% RSLogix 500 project Batch Part Counter.RSS, saved by version 8.30.00.16 %
PROJECT "UNTITLED"    % processor: Bul.1763 MicroLogix 1100 Series B %

PROGRAM FILES
  LAD 2 "MAIN"  7 rungs
  LAD 3 "IO"  5 rungs

DATA FILES
  O0 OUTPUT  5 elements
  I1 INPUT  7 elements
  S2 STATUS  66 elements
  B3 BINARY  1 elements
  T4 TIMER  1 elements
  C5 COUNTER  1 elements
  R6 CONTROL  1 elements
  N7 INTEGER  1 elements
  F8 FLOAT  1 elements

LADDER 2 "MAIN"
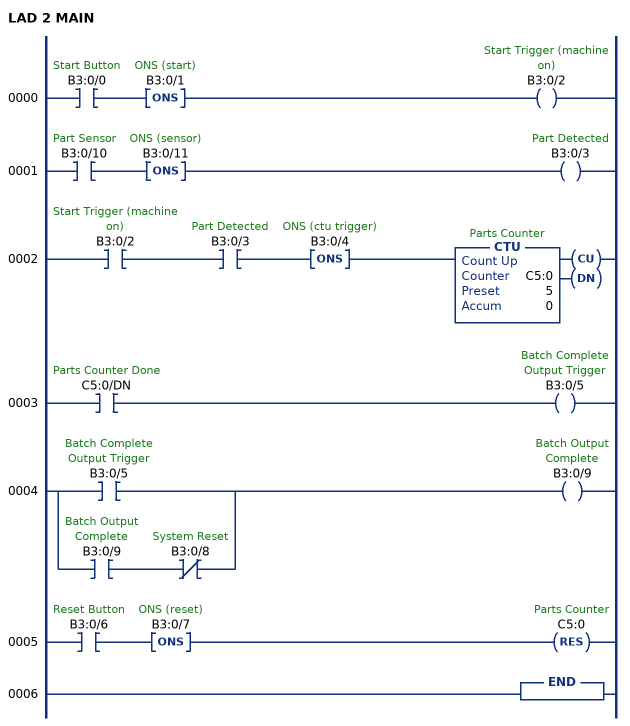
% Rung: 0 %
SOR XIC B3:0/0 ONS B3:0/1 OTE B3:0/2 EOR
%   B3:0/0  "Start Button" %
%   B3:0/1  "ONS (start)" %
%   B3:0/2  "Start Trigger (machine on)" %
% Rung: 1 %
SOR XIC B3:0/10 ONS B3:0/11 OTE B3:0/3 EOR
%   B3:0/10  "Part Sensor" %
%   B3:0/11  "ONS (sensor)" %
%   B3:0/3  "Part Detected" %
% Rung: 2 %
SOR XIC B3:0/2 XIC B3:0/3 ONS B3:0/4 CTU C5:0 5 0 EOR
%   B3:0/2  "Start Trigger (machine on)" %
%   B3:0/3  "Part Detected" %
%   B3:0/4  "ONS (ctu trigger)" %
%   C5:0  "Parts Counter" %
% Rung: 3 %
SOR XIC C5:0/DN OTE B3:0/5 EOR
%   C5:0/DN  "Parts Counter Done" %
%   B3:0/5  "Batch Complete Output Trigger" %
% Rung: 4 %
SOR BST XIC B3:0/5 NXB XIC B3:0/9 XIO B3:0/8 BND OTE B3:0/9 EOR
%   B3:0/5  "Batch Complete Output Trigger" %
%   B3:0/9  "Batch Output Complete" %
%   B3:0/8  "System Reset" %
% Rung: 5 %
SOR XIC B3:0/6 ONS B3:0/7 RES C5:0 EOR
%   B3:0/6  "Reset Button" %
%   B3:0/7  "ONS (reset)" %
%   C5:0  "Parts Counter" %
% Rung: 6 %
SOR END EOR

LADDER 3 "IO"
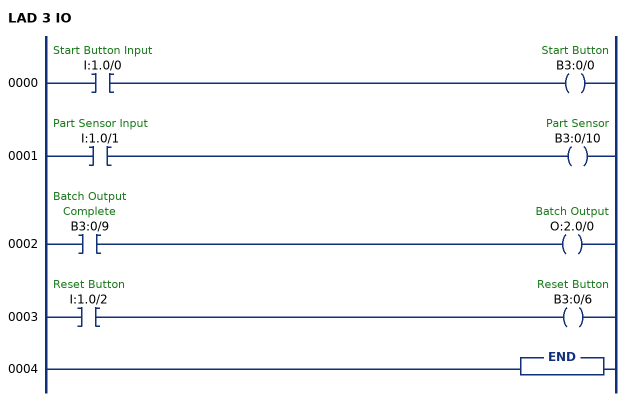
% Rung: 0 %
SOR XIC I:1.0/0 OTE B3:0/0 EOR
%   I:1.0/0  "Start Button Input" %
%   B3:0/0  "Start Button" %
% Rung: 1 %
SOR XIC I:1.0/1 OTE B3:0/10 EOR
%   I:1.0/1  "Part Sensor Input" %
%   B3:0/10  "Part Sensor" %
% Rung: 2 %
SOR XIC B3:0/9 OTE O:2.0/0 EOR
%   B3:0/9  "Batch Output Complete" %
%   O:2.0/0  "Batch Output" %
% Rung: 3 %
SOR XIC I:1.0/2 OTE B3:0/6 EOR
%   I:1.0/2  "Reset Button" %
%   B3:0/6  "Reset Button" %
% Rung: 4 %
SOR END EOR

DATA TABLE (non-zero values as saved)
DATA C5
% .PRE .ACC %
% C5:0 % 5 0
